(* IEC 61131-3 sources: CodesysTest/alpha/export/Pro18_1174_Win10.dev/Plc Logic/Application/Motors/Applied Motion/FB_AppliedMotionStepServoEIPPassthrough.pou, 1 file *)

(* ---- FB_AppliedMotionStepServoEIPPassthrough.pou.st ---- *)
(*#-#-#-#-#-#-#-#-#-#---Declaration---#-#-#-#-#-#-#-#-#-#-#-#-#*)

FUNCTION_BLOCK FB_AppliedMotionStepServoEIPPassthrough EXTENDS FB_AppliedMotionStepServoEIPBase
VAR_INPUT
END_VAR
VAR_OUTPUT
END_VAR
VAR
	homingState : JAW_HOMING_STATES;
	homeRequiredONS : R_TRIG;
	timerHomeDelay : TON;
END_VAR
(*#-#-#-#-#-#-#-#-#-#---Implementation---#-#-#-#-#-#-#-#-#-#-#-#-#*)

SUPER^();
